FUNCTION_BLOCK SC_SecondFloor EXTENDS FB_Chain
VAR_INPUT
	bExecute : BOOL;
	bPlateOpen : BOOL;
END_VAR
VAR_OUTPUT
	bAllPartsPresent: BOOL;	
END_VAR
VAR
	fbPallBeltConveyor : PalletizerConveyor;
	fbPushCyl : Cylinder;
	fbTurnCyl : Cylinder;
	
	fbClampCyl : Cylinder;
	fbClampedSen : Sensor;
	
	fbPusherLimitSen : Sensor;
	fbPresenceDetector : PresenceDetector;
	iCycle : INT;
END_VAR

SUPER^();

fbPushCyl();
fbTurnCyl();

fbClampCyl();
fbPallBeltConveyor();
fbPresenceDetector(bAllPartsPresent => bAllPartsPresent);

METHOD PROTECTED   Busy : BOOL
VAR_INPUT
END_VAR
fbStepWorkerBusy();
CASE fbStepWorkerBusy.uiStep OF
	
	eSecondFloorStart: //send release to scBeltConveyor
	
		iCycle := iCycle + 1;
		IF iCycle = 2
		THEN
			rChainController.releaseForChain('scBeltConveyors', THIS^);
			fbStepWorkerBusy.mNextStep(10);
		ELSE
			fbStepWorkerBusy.mNextStep(20);
		END_IF
		
		
		
	10: //wait for release from scBeltConveyor to start actuators
	
		IF rChainController
			.releaseCheck(THIS^)
			.releaseFromChain(sChainReleasing := 'scBeltConveyors', THIS^)
			.releaseResult(THIS^) 
		THEN
			fbStepWorkerBusy.mNextStep(20);
		END_IF
	
		
	20: //wait for packages
		
		fbTurnCyl.Extend();
		fbPallBeltConveyor.On();
		IF fbPresenceDetector.bAllPartsPresent
		THEN
			bAllPartsPresent := TRUE;
			fbPallBeltConveyor.Off();
			fbStepWorkerBusy.mNextStep(ePushPackages);
		END_IF	
		
	ePushPackages:
	
		fbPushCyl.Extend();
		
		fbStepWorkerBusy
			.mSetTimer(T#2S)
			.mNextStep(eRetractPusher);
		
	eRetractPusher:
	
		fbPushCyl.Retract();
		
		fbStepWorkerBusy
			.mSetTimer(T#2S)
			.mNextStep(eClamp);
			
	eClamp:
	
		fbClampCyl.Extend();
		fbStepWorkerBusy
			.mSetTimer(T#2S)
			.mNextStep(eRetractClamper);
			
	eRetractClamper:
	
		
		fbClampCyl.Retract();
		IF iCycle = 1
		THEN
			fbStepWorkerBusy
				.mSetTimer(T#2S)
				.mNextStep(eSecondFloorStart);
		ELSE
			iCycle := 0;
			fbStepWorkerBusy.mNextStep(eSyncWithFirstFloor);
		END_IF
		
	eSyncWithFirstFloor:
	
		rChainController.releaseForChain('scFirstFloor', THIS^);	
		fbStepWorkerBusy.mNextStep(eWaitForFirstFloor);
	
	eWaitForFirstFloor:
	
		IF rChainController
			.releaseCheck(THIS^)
			.releaseFromChain(sChainReleasing := 'scFirstFloor', THIS^)
			.releaseResult(THIS^) 
		THEN
			fbStepWorkerBusy.mNextStep(eSecondFloorDone);
		END_IF
		
	eSecondFloorDone:
		fbStepWorkerBusy.mNextStep(eSecondFloorStart);
		Done();	
	
END_CASE
END_METHOD

METHOD PROTECTED  Error : BOOL
VAR_INPUT
END_VAR
END_METHOD

METHOD PROTECTED  Idle : BOOL
VAR_INPUT
END_VAR
END_METHOD

METHOD PROTECTED  Init : BOOL
VAR_INPUT
END_VAR
Start();
END_METHOD

METHOD PROTECTED  Prepare : BOOL
VAR_INPUT
END_VAR
END_METHOD

METHOD PROTECTED  Ready : BOOL
VAR_INPUT
END_VAR

fbStepWorkerReady();
CASE fbStepWorkerReady.uiStep OF
	
	0: 
	
		IF bExecute THEN
			fbStepWorkerReady.mNextStep(10);
		END_IF
		
	10:
		
		IF NOT fbPresenceDetector.bAllPartsPresent
			AND NOT bPlateOpen
		THEN
			rChainController.releaseForChain('scBeltConveyors', THIS^);	
			fbStepWorkerReady.mNextStep(20);	
		END_IF
	
	20:
		
		IF rChainController
			.releaseCheck(THIS^)
			.releaseFromChain(sChainReleasing := 'scBeltConveyors', THIS^)
			.releaseResult(THIS^) 
		THEN
			fbStepWorkerReady.mNextStep(0);
			Execute();
		END_IF
		
END_CASE
END_METHOD

METHOD PROTECTED  Waiting : BOOL
VAR_INPUT
END_VAR
END_METHOD

END_FUNCTION_BLOCK

(* stored: Version 1.1.0.1, ProductVersion 3.1.4024.2
   POU SC_SecondFloor: Id {cbbd2891-fc43-4186-abe0-a1a8275dd971}, SpecialFunc None
   Method Busy: Id {9ab5514a-a41d-490b-9a99-ffb6abe5f8ac}
   Method Error: Id {54fc011b-0bdc-497c-83e9-e16b470645fb}
   Method Idle: Id {f1b86f65-2ab3-4c06-9c94-6ef43dc472ea}
   Method Init: Id {97c84f6f-0187-4362-810c-4de0217e8b37}
   Method Prepare: Id {36c933cf-9b53-4ec2-b3d1-14bbe5df98f2}
   Method Ready: Id {517c8a14-559f-4f37-8a25-7a64b054a837}
   Method Waiting: Id {97c5ccd7-d726-4b89-af53-2743cec1a3bc} *)
